FUNCTION_BLOCK PlantFB (* Composite Function Block Type *)
  (* Standard: 61499-2 *)
  (* Version 1.0, 2019-03-19, Duc Do Tran, OFFIS e.V. *)
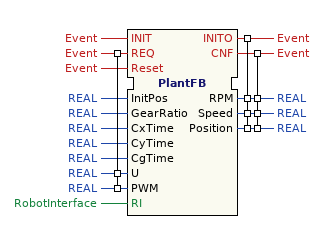
  EVENT_INPUT
    INIT;
    REQ WITH U, PWM;
    Reset;
  END_EVENT
  EVENT_OUTPUT
    INITO WITH Position, Speed, RPM;
    CNF WITH Position, Speed, RPM; (* Execution Confirmation *)
  END_EVENT
  VAR_INPUT
    InitPos : REAL := 0;
    GearRatio : REAL := 0.1;
    CxTime : REAL := 0.35;
    CyTime : REAL := 0.18;
    CgTime : REAL := 0.09;
    U : REAL := 24;
    PWM : REAL;
  END_VAR
  VAR_OUTPUT
    RPM : REAL;
    Speed : REAL;
    Position : REAL := 180; (* Output event qualifier *)
  END_VAR
  SOCKETS
    RI : RobotInterface; (* AdapterType *)
  END_SOCKETS
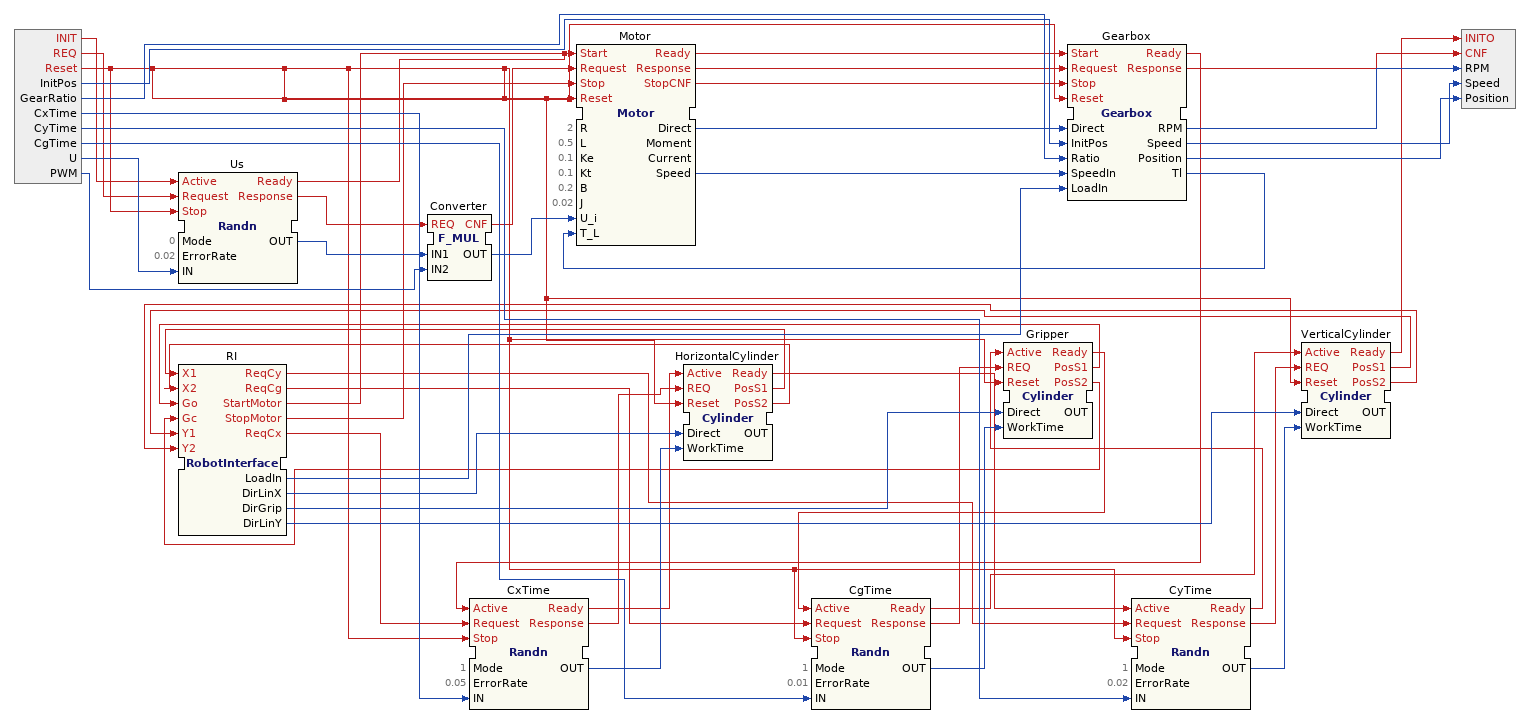
  FBS
    Converter : F_MUL;
    Us : Randn(Mode := 0, ErrorRate := 0.02);
    CyTime : Randn(Mode := 1, ErrorRate := 0.02);
    CgTime : Randn(Mode := 1, ErrorRate := 0.01);
    Motor : Motor(R := 2, L := 0.5, Ke := 0.1, Kt := 0.1, B := 0.2, J := 0.02);
    Gearbox : Gearbox;
    CxTime : Randn(Mode := 1, ErrorRate := 0.05);
    HorizontalCylinder : Cylinder;
    Gripper : Cylinder;
    VerticalCylinder : Cylinder;
  END_FBS
  EVENT_CONNECTIONS
    INIT TO Us.Active;
    REQ TO Us.Request;
    Us.Response TO Converter.REQ;
    RI.ReqCy TO CyTime.Request;
    RI.ReqCg TO CgTime.Request;
    RI.StartMotor TO Motor.Start;
    Converter.CNF TO Motor.Request;
    RI.StopMotor TO Motor.Stop;
    Reset TO Motor.Reset;
    Motor.Ready TO Gearbox.Start;
    Motor.StopCNF TO Gearbox.Stop;
    Reset TO Gearbox.Reset;
    Gearbox.Response TO CNF;
    Motor.Response TO Gearbox.Request;
    Gearbox.Ready TO CxTime.Active;
    RI.ReqCx TO CxTime.Request;
    CxTime.Ready TO HorizontalCylinder.Active;
    CxTime.Response TO HorizontalCylinder.REQ;
    HorizontalCylinder.Ready TO CyTime.Active;
    HorizontalCylinder.PosS1 TO RI.X1;
    HorizontalCylinder.PosS2 TO RI.X2;
    CyTime.Ready TO Gripper.Active;
    CgTime.Response TO Gripper.REQ;
    Gripper.Ready TO CgTime.Active;
    Gripper.PosS1 TO RI.Go;
    Gripper.PosS2 TO RI.Gc;
    CgTime.Ready TO VerticalCylinder.Active;
    CyTime.Response TO VerticalCylinder.REQ;
    VerticalCylinder.Ready TO INITO;
    VerticalCylinder.PosS1 TO RI.Y1;
    VerticalCylinder.PosS2 TO RI.Y2;
    Reset TO HorizontalCylinder.Reset;
    Reset TO Gripper.Reset;
    Reset TO VerticalCylinder.Reset;
    Us.Ready TO Motor.Start;
    Reset TO Us.Stop;
    Reset TO CxTime.Stop;
    Reset TO CgTime.Stop;
    Reset TO CyTime.Stop;
  END_CONNECTIONS
  DATA_CONNECTIONS
    U TO Us.IN;
    Us.OUT TO Converter.IN1;
    CyTime TO CyTime.IN;
    CgTime TO CgTime.IN;
    PWM TO Converter.IN2;
    Converter.OUT TO Motor.U_i;
    InitPos TO Gearbox.InitPos;
    GearRatio TO Gearbox.Ratio;
    Motor.Speed TO Gearbox.SpeedIn;
    RI.LoadIn TO Gearbox.LoadIn;
    Gearbox.RPM TO RPM;
    Gearbox.Speed TO Speed;
    Gearbox.Position TO Position;
    Gearbox.Tl TO Motor.T_L;
    Motor.Direct TO Gearbox.Direct;
    CxTime TO CxTime.IN;
    RI.DirLinX TO HorizontalCylinder.Direct;
    CxTime.OUT TO HorizontalCylinder.WorkTime;
    RI.DirGrip TO Gripper.Direct;
    CgTime.OUT TO Gripper.WorkTime;
    RI.DirLinY TO VerticalCylinder.Direct;
    CyTime.OUT TO VerticalCylinder.WorkTime;
  END_CONNECTIONS
END_FUNCTION_BLOCK
